{attribute 'hide'}
{attribute clr [ExcludeFromApiDocumentation()]}
FUNCTION_BLOCK ABSTRACT _internals_TcoContext EXTENDS TcoContext
VAR
	_probeCurrentCycleCount  : ULINT;	
	_probeRunRequiredCycles : ULINT;
	_testId : ULINT;
	_testDoneCounter : ULINT;
	_plcCycleCounter : ULINT;
END_VAR

{attribute 'TcRpcEnable'}
METHOD PROTECTED FINAL _Close
THIS^.Close();
END_METHOD

METHOD _GetSynchParams : RtcSynchParams
_GetSynchParams := RtcPrg._RtcSynchParams;
END_METHOD

{attribute 'TcRpcEnable'}
METHOD PROTECTED FINAL _Open
THIS^.Open();
END_METHOD

{attribute 'TcRpcEnable'}
METHOD PROTECTED FINAL _rtcUpdate
THIS^._rtc.UpdateInternal();
END_METHOD

METHOD ClearPlcCycleCounter
_plcCycleCounter := 0;
END_METHOD

METHOD ClearTestDoneCounter
_testDoneCounter := 0;
END_METHOD

METHOD ProbeDoneWhen
VAR_INPUT
	inCondition : BOOL;
END_VAR
IF inCondition THEN
    _testDoneCounter := _testDoneCounter + 1;
    _probeRunRequiredCycles := 0;
    _probeCurrentCycleCount := 0;
	{warning disable C0195}
    _testId := -1;
	{warning enable C0195}
END_IF
END_METHOD

METHOD ProbeRun
IF(_probeCurrentCycleCount < _probeRunRequiredCycles) THEN 
	_plcCycleCounter := _plcCycleCounter + 1;
	SUPER^.Run();	
	_probeCurrentCycleCount := _probeCurrentCycleCount + 1;
END_IF;
END_METHOD

END_FUNCTION_BLOCK

(* stored: Version 1.1.0.1
   POU _internals_TcoContext: Id {0c059046-c7d3-0372-268c-dca3da778e0c}, SpecialFunc None
   Method _Close: Id {e2e1d492-d989-0bc8-0108-b8347f5c2d4e}
   Method _GetSynchParams: Id {e3cf5488-c586-0883-2979-a24e3d4feb8c}
   Method _Open: Id {d83dfe53-3a8f-0733-3457-8d9db7cfe99c}
   Method _rtcUpdate: Id {cb574abf-9f5d-03d2-0459-a21349c4ee2b}
   Method ClearPlcCycleCounter: Id {c583d8a3-29fc-0453-3825-9f103d525599}
   Method ClearTestDoneCounter: Id {28fd480f-5bde-063d-3077-fc93368b2e04}
   Method ProbeDoneWhen: Id {a83a1f55-5d29-0fd3-0d4c-5249b5104c8a}
   Method ProbeRun: Id {98c82b04-49c1-0249-2482-4f11240daf4e} *)
